{attribute 'qualified_only'}
VAR_GLOBAL
	Cycle_Start:BOOL;
	Cycle_Stop:BOOL;
	AutoMode:BOOL;
	ManualMode:BOOL;
	Estop:BOOL;
	Reset:BOOL;
	
END_VAR

(* stored: Version 1.1.0.1, ProductVersion 3.1.4024.16
   GVL HMI: Id {e9b51b3d-2f7f-46c3-a0ea-346b3789bb74} *)
